				fbADSWRITE( WRITE:= FALSE );
				fbADSWRITE(
					NETID:= TcMcGlobal.NCNETID_TCMC,
					PORT:= AMSPORT_R0_NCSAF,
					IDXGRP:= 16#4200 + Axis.NcToPlc.AxisId,
					IDXOFFS:= 16#63,
					LEN:= SIZEOF(stWriteDriveOperationMode),
					SRCADDR:= ADR(stWriteDriveOperationMode),
					WRITE:= TRUE,
					TMOUT:= TcMcGlobal.tADSTimeOut);
				state := STATE_ORDER;
			END_IF
		END_IF

	STATE_ORDER :
		fbADSWRITE();
		IF NOT fbADSWRITE.BUSY THEN
			IF NOT fbADSWRITE.ERR THEN
				Done := TRUE;
			ELSE
				Error := TRUE;
				ErrorID := fbADSWRITE.ERRID;
			END_IF
			state := STATE_INITIALIZATION;
		END_IF

END_CASE

ADSbusy := fbADSWRITE.BUSY;
IF state = STATE_INITIALIZATION THEN
	(* reset Busy immediately  when sequence ends *)
	IF Busy THEN
		LastExecutionResult.Done := Done;
		LastExecutionResult.Error := Error;
		LastExecutionResult.ErrorID := ErrorID;
	END_IF
	Busy := FALSE;
END_IF

END_FUNCTION_BLOCK

// POUs/Administrative/Extensions/MC_CalcDynamicsByRampTime
FUNCTION_BLOCK MC_CalcDynamicsByRampTime
VAR_INPUT
	Velocity 	: LREAL;		// must be greaater than zero
	RampTime 	: LREAL;		// must be greaater than zero
	Stiffness 	: LREAL := 0.5;	// range 0..1.0 (will be silently reduced to 0.99 if 0.99 < Stiffness <= 1.0) 
END_VAR
VAR_OUTPUT
	Error 		: BOOL;
	ErrorID 	: UDINT;
	Acceleration: LREAL;	
	Deceleration: LREAL;	// identical to Acceleration !	
	Jerk 		: LREAL;
END_VAR
VAR
	t1: LREAL;	// time of jerk to ramp up to constant acceleration
	t2: LREAL;	// time of constant acceleration
	TriggerExecute: R_trig;
END_VAR

// Description:
//
// The function block calculates Acceleration and Jerk values to ramp up to a defined Velcoity in a defined RampTime.
// The calculation assumes that the Velocity can be reached (long distance moves). The calculated dynamics can be  
// used on short distances moves as well but the ramp up time will then be shorter. 
//
// Velocity : Velocity value to ramp up to during RampTime
// RampTime : time to ramp up to Velocity
// Stiffness: = time of constant acceleration / time to ramp up to constant acceleration (jerk time)
// 		Sample:  
// 			Stiffness = 0.0	: triangular acceleration profile
// 			Stiffness = 0.5	: trapezoid acceleration profile with time of constant acceleration = 1/3 RampTime
//			Stiffness = 1.0	: rectangular acceleration profile 

// check input parameters
IF stiffness<0 OR stiffness>1.0 OR RampTime<0.001 OR Velocity < 0.001 THEN
	// error
	Error := TRUE;
	ErrorID := MC_ERROR_PARAMETER_NOT_CORRECT;
	Acceleration := 0;
	Deceleration := 0;
	Jerk := 0;
	RETURN;
END_IF

// silent reduction of Stiffness between 0.99 and 1.0 
IF Stiffness > 0.99 THEN
	Stiffness:=0.99;
END_IF

// t1 = time of jerk to ramp up to constant acceleration
t1 := (1-Stiffness) / (2-Stiffness) * RampTime; 
(*
// check ?
IF t1<0.000250 THEN
	t1 := 0.000250;
END_IF
*)
// t2 = time of constant acceleration
t2 := RampTime - t1 - t1; // RampTime - 2*t1	

Acceleration := Velocity / (t1 + t2);
Deceleration := Acceleration;
Jerk := Acceleration / t1;

Error := FALSE; // result okay
ErrorID := 0;

END_FUNCTION_BLOCK

// POUs/Administrative/Extensions/MC_SelectControlLoop
{attribute 'conditionalshow_all_locals'}
FUNCTION_BLOCK MC_SelectControlLoop
VAR_IN_OUT
	Axis : AXIS_REF; (*Reference to an axis*)
END_VAR
VAR_INPUT
	Execute : BOOL;
	EncoderIndex : UINT;
	SelectType : E_SelectControlLoopType;
	SyncValue : LREAL;
	ExtSetPointGen : BOOL;
END_VAR
VAR_OUTPUT
	Done : BOOL;
	Busy : BOOL;
	Error : BOOL;
{attribute 'displaymode':='hex'}
	ErrorID : UDINT;
END_VAR
VAR
	LastExecutionResult: 	_ST_FunctionBlockResults;
	ADSbusy: BOOL;
	state: _E_TcMC_STATES := STATE_INITIALIZATION;
	stSelectControlLoop : ST_SelectControlLoop;
	fbADSWRITE: ADSWRITE;
END_VAR
VAR
	TriggerExecute: R_TRIG;
END_VAR

TriggerExecute(CLK:=Execute);

CASE state OF
	STATE_INITIALIZATION :
		Busy := FALSE;
		IF NOT Execute THEN
			Done := FALSE;
			Error := FALSE;
			ErrorID := 0;
		END_IF
		IF TriggerExecute.Q THEN
			Busy := TRUE;

			LastExecutionResult.Done := FALSE;
			LastExecutionResult.CommandAborted := FALSE;
			LastExecutionResult.Error := FALSE;
			LastExecutionResult.ErrorID := 0;
	
			stSelectControlLoop.EncoderIndex := EncoderIndex;
			stSelectControlLoop.SelectType := SelectType;
			stSelectControlLoop.SyncValue := SyncValue;
			stSelectControlLoop.ExtSetPointGen := SEL(ExtSetPointGen, 0 ,1);

			fbADSWRITE( WRITE:= FALSE );
			fbADSWRITE(
				NETID:= TcMcGlobal.NCNETID_TCMC,
				PORT:= TcMcGlobal.NCPORT_TCMC,
				IDXGRP:= 16#4200 + Axis.NcToPlc.AxisId,
				IDXOFFS:= 16#52,
				LEN:= SIZEOF(stSelectControlLoop),
				SRCADDR:= ADR(stSelectControlLoop),
				WRITE:= TRUE,
				TMOUT:= TcMcGlobal.tADSTimeOut);
			state := STATE_ORDER;
		END_IF

	STATE_ORDER :
		fbADSWRITE();
		IF NOT fbADSWRITE.BUSY THEN
			IF NOT fbADSWRITE.ERR THEN
				Done := TRUE;
			ELSE
				Error := TRUE;
				ErrorID := fbADSWRITE.ERRID;
			END_IF
			state := STATE_INITIALIZATION;
		END_IF

END_CASE

ADSbusy := fbADSWRITE.BUSY;
IF state = STATE_INITIALIZATION THEN
	(* reset Busy immediately  when sequence ends *)
	IF Busy THEN
		LastExecutionResult.Done := Done;
		LastExecutionResult.Error := Error;
		LastExecutionResult.ErrorID := ErrorID;
	END_IF
	Busy := FALSE;
END_IF

END_FUNCTION_BLOCK

// POUs/Administrative/Extensions/MC_WriteNcIoOutput
{attribute 'conditionalshow_all_locals'}
FUNCTION_BLOCK MC_WriteNcIoOutput
VAR_IN_OUT
	Axis				: AXIS_REF;
END_VAR
VAR_INPUT
	Execute				: BOOL;

	Device				: E_NcIoDevice := NcIoDeviceDrive;	
	NcIoOutput			: E_NcIoOutput := NcIoOutputnCtrl1;
	
	BitSelectMask		: UDINT := 16#0;
	BitValues			: UDINT;
END_VAR
VAR_OUTPUT
	Done				: BOOL;
	Busy				: BOOL;
	Error				: BOOL;
{attribute 'displaymode':='hex'}
	ErrorId				: UDINT;
END_VAR
VAR
	FlExecute			: R_TRIG;
	
	State				: UDINT;
	
	ReadDriveAddress	: MC_ReadDriveAddress;
	DriveAddress		: ST_DriveAddress;
	
	AdsWrite			: ADSWRITE;
	IdxGrp				: UDINT;

	NcIoOutputData		: _ST_NcIoOutputData;
END_VAR

FlExecute(CLK:=Execute);

CASE State OF
	0:
		IF NOT Execute THEN
			Done := FALSE;
			Busy := FALSE;
			Error := FALSE;
			ErrorId := 0;
		END_IF
		
		IF FlExecute.Q THEN
			Busy := TRUE;
			IF DriveAddress.NcAxisId = Axis.NcToPlc.AxisId THEN
				State := State + 2;
			ELSE
				State := State + 1;
			END_IF
		END_IF
		
	1: // Read drive address
		ReadDriveAddress(
			Axis			:= Axis, 
			Execute			:= TRUE, 
			DriveAddress	=> DriveAddress);

		IF NOT ReadDriveAddress.Busy AND ReadDriveAddress.Done THEN
			ReadDriveAddress(
				Axis			:= Axis, 
				Execute			:= FALSE); 

			State := State + 1	;		
		ELSIF NOT ReadDriveAddress.Busy AND ReadDriveAddress.Error THEN
			Busy := FALSE;
			Error := TRUE;
			ErrorId := ReadDriveAddress.ErrorID;
			
			ReadDriveAddress(
				Axis			:= Axis, 
				Execute			:= FALSE); 
				
			State := 0;	
		END_IF

	2: // Write nc io output
		CASE Device OF
			NcIoDeviceDrive:
				IdxGrp := 16#7300 + DriveAddress.NcDriveId;				
			NcIoDeviceEncoder:
				IdxGrp := 16#5300 + DriveAddress.NcEncoderId;				
			ELSE
				Busy := FALSE;
				Error := TRUE;
				ErrorId := 16#4B06;

				State := 0;
				RETURN;				
		END_CASE
	
		CASE NcIoOutput OF
			NcIoOutputnCtrl1:
				NcIoOutputData.ByteOffset := 16#08;
			NcIoOutputnCtrl2:
				NcIoOutputData.ByteOffset := 16#09;
			NcIoOutputnCtrl3:
				NcIoOutputData.ByteOffset := 16#0A;
			NcIoOutputnCtrl4:
				NcIoOutputData.ByteOffset := 16#0B;
			NcIoOutputnCtrl5:
				NcIoOutputData.ByteOffset := 16#1C;
			NcIoOutputnCtrl6:
				NcIoOutputData.ByteOffset := 16#1D;
			NcIoOutputnCtrl7:
				NcIoOutputData.ByteOffset := 16#1E;
			NcIoOutputnCtrl8:
				NcIoOutputData.ByteOffset := 16#1F;
			NcIoOutputnDataOut1:
				NcIoOutputData.ByteOffset := 16#00;
			NcIoOutputnDataOut2:
				NcIoOutputData.ByteOffset := 16#04;
			NcIoOutputnDataOut3:
				NcIoOutputData.ByteOffset := 16#0C;
			NcIoOutputnDataOut4:
				NcIoOutputData.ByteOffset := 16#10;
			NcIoOutputnDataOut5:
				NcIoOutputData.ByteOffset := 16#14;
			NcIoOutputnDataOut6:
				NcIoOutputData.ByteOffset := 16#18;
			ELSE			
				Busy := FALSE;
				Error := TRUE;
				ErrorId := 16#4B06;

				State := 0;
				RETURN;				
		END_CASE

		NcIoOutputData.BitSelectMask 	:= BitSelectMask;
		NcIoOutputData.BitValues		:= BitValues;

		AdsWrite(
			NETID			:= '', 
			PORT			:= 501, 
			IDXGRP			:= IdxGrp, 
			IDXOFFS			:= 16#01, 
			LEN				:= SIZEOF(NcIoOutputData), 
			SRCADDR			:= ADR(NcIoOutputData), 
			WRITE			:= TRUE, 
			TMOUT			:= T#5S); 

		IF AdsWrite.BUSY THEN
			State := State + 1;
		END_IF

	3: // wait for result
		AdsWrite();

		IF NOT AdsWrite.BUSY THEN
			IF NOT AdsWrite.ERR THEN
				Done := TRUE;				
			ELSE
				Error := TRUE;
				ErrorId := AdsWrite.ERRID;				
			END_IF
			Busy := FALSE;
			
			AdsWrite(WRITE := FALSE);
			
			State := 0;
		END_IF
END_CASE

END_FUNCTION_BLOCK

// POUs/Administrative/Status and Parameter/MC_ReadActualPosition
FUNCTION_BLOCK MC_ReadActualPosition
(*	This Function Block returns the actual position. *)
VAR_IN_OUT
	Axis			:	AXIS_REF; (*Reference to an axis*)
END_VAR
VAR_INPUT
	Enable		:	BOOL;		
END_VAR
VAR_OUTPUT
	Valid		:	BOOL;		
	Busy		:	BOOL;		
	Error		:	BOOL;	
{attribute 'displaymode':='hex'}
	ErrorID		:	UDINT;	
	Position		:	LREAL;		
END_VAR
VAR
END_VAR

Error := FALSE;
ErrorID := 0;
IF Enable THEN
	Busy := TRUE;
	Position := Axis.NcToPlc.ActPos;
	Valid := TRUE;
ELSE
	Busy := FALSE;
	Position := 0.0;
	Valid := FALSE;
END_IF;

END_FUNCTION_BLOCK

// POUs/Administrative/Status and Parameter/MC_ReadActualVelocity
FUNCTION_BLOCK MC_ReadActualVelocity
(*
	This Function Block returns the value of the actual velocity as long as Enable is 
	set. Valid is true when the data-output ActualVelocity is valid. If Enable is reset, the 
	data loses its validity, and all outputs are reset, no matter if new data is available.
*)
VAR_IN_OUT
	Axis			:	AXIS_REF; (*Reference to an axis*)
END_VAR
VAR_INPUT
	Enable 		: 	BOOL;	
END_VAR
VAR_OUTPUT
	Valid 		: 	BOOL;	
	Busy 		: 	BOOL;	
	Error 		: 	BOOL;	
{attribute 'displaymode':='hex'}
	ErrorID 		: 	UDINT;	
	ActualVelocity (* Velocity *): 	LREAL;	
END_VAR
VAR
END_VAR

Error := FALSE;
ErrorID := 0;
IF Enable THEN
	Busy := TRUE;
	Valid := TRUE;
	ActualVelocity := Axis.NcToPlc.ActVelo;
ELSE
	Busy := FALSE;
	Valid := FALSE;
	ActualVelocity := 0;
END_IF

END_FUNCTION_BLOCK

// POUs/Administrative/Status and Parameter/MC_ReadAxisError
FUNCTION_BLOCK MC_ReadAxisError
(*
	This Function Block presents general axis errors not relating to the Function Blocks. 
	(for instance axis errors, drive errors, communication errors)
 *)
VAR_IN_OUT
	Axis				:	AXIS_REF; (*Reference to an axis*)
END_VAR
VAR_INPUT
	Enable			:	BOOL;		
END_VAR
VAR_OUTPUT
	Valid			:	BOOL;		
	Busy			:	BOOL;		
	Error			:	BOOL;	
{attribute 'displaymode':='hex'}
	ErrorID			:	DWORD;	
	AxisErrorID		:	DWORD;	
END_VAR
VAR
END_VAR

IF Enable THEN
	Busy		 := TRUE;
	Valid 		:=  TRUE;
	ErrorID 		:= 0;
	AxisErrorID 	:= Axis.NcToPlc.ErrorCode;
	Error		:= ErrorID <> 0;
ELSE
	Busy 		:= FALSE;
	Valid 		:= FALSE;
	Error 		:= FALSE;	(* reset at falling edge of Execute *)
	ErrorID 		:= 0;
	AxisErrorID 	:= 0;
END_IF;

END_FUNCTION_BLOCK

// POUs/Administrative/Status and Parameter/MC_WriteBoolParameter
FUNCTION_BLOCK MC_WriteBoolParameter
(*	This Function Block modifies the value of a vendor specific boolean parameter. *)
VAR_IN_OUT
	Axis				:	AXIS_REF; (*Reference to an axis*)
END_VAR
VAR_INPUT
	Execute			:	BOOL;	
	ParameterNumber	:	MC_AxisParameter; // 2023-03 KSt changed from INT to MC_AxisParameter	
	Value			:	BOOL;	
(* 	ExecutionMode 	: 	MC_EXECUTION_MODE *)		(* not available *)
END_VAR
VAR_OUTPUT
	Done			:	BOOL;	
	Busy			: 	BOOL;
	Error			:	BOOL;	
{attribute 'displaymode':='hex'}
	ErrorID			:	UDINT;	
END_VAR
VAR
	ADSbusy		: 	BOOL;
	fbReadWriteParameter: 	_FB_ReadWriteParameter;
END_VAR
VAR
//{attribute 'conditionalshow'}
//	nParatype 		:	_E_ParameterType;	(* removed 2021-04-12 KSt - not required *)
{attribute 'conditionalshow'}
	dwValue 			: 	DWORD;
{attribute 'conditionalshow'}
	lrValue 			: 	LREAL;
{attribute 'conditionalshow'}
	fbTrigger 		: 	R_TRIG;
END_VAR

IF NOT Execute THEN
	Done := FALSE;
	Error := FALSE;			(* reset at falling edge of Execute *)
	ErrorID := 0;
END_IF
fbTrigger(CLK:= Execute);
IF fbTrigger.Q AND NOT Busy THEN
	Busy := TRUE;
	Done := FALSE;
	Error := FALSE;
	ErrorID := MC_ERROR_NO_ERROR;
END_IF;
(* *)
IF Busy THEN
//	nParatype := PARAMETERTYPE_BOOL;
	fbReadWriteParameter.ParameterPointer := 0;
	fbReadWriteParameter.ParameterSize := 0;
	fbReadWriteParameter(Enable:= TRUE, ParameterNumber:= ParameterNumber, Mode:= READWRITEPARAMETERMODE_WRITE,
						(*ParameterType:=nParatype,*) Axis:= Axis, ValueLreal:= lrValue, ValueDword := dwValue, ValueBool := Value);
	IF fbReadWriteParameter.Done THEN
		Done := TRUE;
		Busy := FALSE;
		fbReadWriteParameter(Enable:= FALSE, ParameterNumber:= ParameterNumber, Mode:= READWRITEPARAMETERMODE_WRITE,
						(*ParameterType:= nParatype,*) Axis:= Axis, ValueLreal:= lrValue, ValueDword := dwValue, ValueBool := Value);
	END_IF;
	IF fbReadWriteParameter.Error THEN
		Busy := FALSE;
		Done := FALSE;
		Error := TRUE;
		ErrorID := fbReadWriteParameter.ErrorID;
		fbReadWriteParameter(Enable:= FALSE, ParameterNumber:= ParameterNumber, Mode:= READWRITEPARAMETERMODE_WRITE,
						(*ParameterType:= nParatype,*) Axis:= Axis, ValueLreal:= lrValue, ValueDword := dwValue, ValueBool := Value);
	END_IF;
END_IF;

ADSbusy := fbReadWriteParameter.ADSbusy;

END_FUNCTION_BLOCK

// POUs/Administrative/Status and Parameter/MC_WriteLargeParameter
FUNCTION_BLOCK MC_WriteLargeParameter
(*	This Function Block modifies the value of a vendor specific parameter. *)
VAR_IN_OUT
	Axis				:	AXIS_REF; (*Reference to an axis*)
END_VAR
VAR_INPUT
	Execute			:	BOOL;	
	ParameterNumber	:	MC_AxisParameter; // 2023-03 KSt changed from INT to MC_AxisParameter		
//	Value			:	LREAL;	
	ParameterPointer: 	PVOID;	// for structured parameters - KSt 2021-03-04
	ParameterSize	:	USINT; 	// for structured parameters  - KSt 2021-03-04
(* 	ExecutionMode 	: 	MC_EXECUTION_MODE *)	(* not available *)
END_VAR
VAR_OUTPUT
	Done			:	BOOL;		
	Busy			: 	BOOL;		
	Error			:	BOOL;		
{attribute 'displaymode':='hex'}
	ErrorID			:	UDINT;		
END_VAR
VAR
	ADSbusy			: 	BOOL;
	fbReadWriteParameter: _FB_ReadWriteParameter;
END_VAR
VAR
{attribute 'conditionalshow'}
	lrValue 		: 	LREAL;
{attribute 'conditionalshow'}
	dwValue 		: 	DWORD;
{attribute 'conditionalshow'}
	bValue 			: 	BOOL;
{attribute 'conditionalshow'}
	fbTrigger 		: 	R_TRIG;
END_VAR

IF NOT Execute THEN
	Done := FALSE;
	Error := FALSE;			(* reset at falling edge of Execute *)
	ErrorID := 0;
END_IF
fbTrigger(CLK:= Execute);
IF fbTrigger.Q AND NOT Busy THEN
	Busy := TRUE;
	Done := FALSE;
	Error := FALSE;
	ErrorID := MC_ERROR_NO_ERROR;
END_IF;
(* *)
IF Busy THEN
	fbReadWriteParameter.ParameterPointer := 0;
	fbReadWriteParameter.ParameterSize := 0;
	fbReadWriteParameter(Enable:= TRUE, ParameterNumber:= ParameterNumber, Mode:= READWRITEPARAMETERMODE_WRITE,
						Axis:= Axis, ValueLreal:= lrValue, ValueDword := dwValue, ValueBool := bValue,
						ParameterPointer := ParameterPointer, ParameterSize:=ParameterSize); 
	IF fbReadWriteParameter.Done THEN
		Done := TRUE;
		Busy := FALSE;
		fbReadWriteParameter(Enable:= FALSE, ParameterNumber:= ParameterNumber, Mode:= READWRITEPARAMETERMODE_WRITE,
							Axis:= Axis, ValueLreal:= lrValue, ValueDword := dwValue, ValueBool := bValue,
							ParameterPointer := ParameterPointer, ParameterSize:=ParameterSize); 
	END_IF;
	IF fbReadWriteParameter.Error THEN
		Busy := FALSE;
		Done := FALSE;
		Error := TRUE;
		ErrorID := fbReadWriteParameter.ErrorID;
		fbReadWriteParameter(Enable:= FALSE, ParameterNumber:= ParameterNumber, Mode:= READWRITEPARAMETERMODE_WRITE,
							Axis:= Axis, ValueLreal:= lrValue, ValueDword := dwValue, ValueBool := bValue,
							ParameterPointer := ParameterPointer, ParameterSize:=ParameterSize); 
	END_IF;
END_IF;

ADSbusy := fbReadWriteParameter.ADSbusy;

END_FUNCTION_BLOCK

// POUs/Administrative/Status and Parameter/MC_WriteLargeParameterPersistent
FUNCTION_BLOCK MC_WriteLargeParameterPersistent
VAR_IN_OUT
	Axis: AXIS_REF; (*Reference to an axis*)
END_VAR
VAR_INPUT
	Execute			: BOOL;
	ParameterNumber	: MC_AxisParameter; // 2023-03 KSt changed from INT to MC_AxisParameter
//	Value: LREAL;
	ParameterPointer: 	PVOID;	// for structured parameters - KSt 2021-03-04
	ParameterSize	:	USINT; 	// for structured parameters  - KSt 2021-03-04
END_VAR
VAR_OUTPUT
	Done: BOOL;
	Busy: BOOL;
	Error: BOOL;
{attribute 'displaymode':='hex'}
	ErrorID: UDINT;
END_VAR
VAR
	fbWriteParameterPersistent: _FB_WriteParameterPersistent;
END_VAR

fbWriteParameterPersistent(
	Axis:= Axis, 
	Execute:= Execute, 
	ParameterNumber:= ParameterNumber, 
//	Value:= Value, 
	ParameterPointer := ParameterPointer, 
	ParameterSize:=ParameterSize,
	Done=> Done, 
	Busy=> Busy, 
	Error=> Error, 
	ErrorID=> ErrorID);

END_FUNCTION_BLOCK

// POUs/Motion/Phasing/MC_HaltPhasing
FUNCTION_BLOCK MC_HaltPhasing
VAR_IN_OUT
	Master 			: 	AXIS_REF; (*Reference to an axis*)
	Slave 			: 	AXIS_REF; (*Reference to an axis*)
END_VAR
VAR_INPUT
	Execute			:	BOOL;		(* Start the motion at rising edge *)
	Deceleration	:	LREAL;		(* Value of the maximum deceleration *)
	Jerk			:	LREAL;		(* Value of the maximum jerk *)
	BufferMode		:	MC_BufferMode;	
	Options			: 	ST_PhasingOptions;		(* optional parameters *)
END_VAR
VAR_OUTPUT
	Done			:	BOOL;	
	Busy			: 	BOOL;	
	Active			: 	BOOL;	
	CommandAborted	:	BOOL;	
	Error			:	BOOL;	
{attribute 'displaymode':='hex'}
	ErrorID			:	UDINT;	
END_VAR

VAR
	PhasingGeneric : _FB_PhasingGeneric;
END_VAR

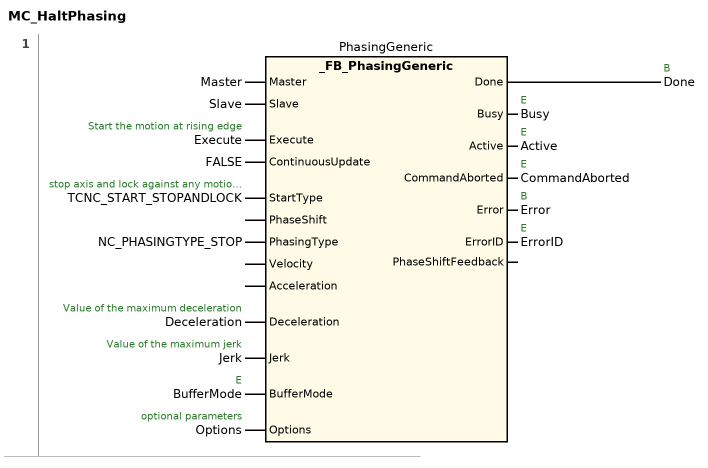
// NETWORK 1
//   Execute: Start the motion at rising edge
//   TCNC_START_STOPANDLOCK: stop axis and lock against any motion commands
//   Deceleration: Value of the maximum deceleration
//   Jerk: Value of the maximum jerk
//   BufferMode: E
//   Options: optional parameters
//   Busy: E
//   Active: E
//   CommandAborted: E
//   Error: B
//   ErrorID: E
//   Done: B
PhasingGeneric(
    Master := Master,
    Slave := Slave,
    Execute := Execute,
    ContinuousUpdate := FALSE,
    StartType := TCNC_START_STOPANDLOCK,
    PhasingType := NC_PHASINGTYPE_STOP,
    Deceleration := Deceleration,
    Jerk := Jerk,
    BufferMode := BufferMode,
    Options := Options,
    Busy => Busy,
    Active => Active,
    CommandAborted => CommandAborted,
    Error => Error,
    ErrorID => ErrorID); // _FB_PhasingGeneric
Done := PhasingGeneric.Done;

END_FUNCTION_BLOCK

// POUs/Motion/Phasing/MC_PhasingAbsolute
(*	This Function Block creates an absolute phase shift in the master position of a slave axis. 
	The master position is shifted in relation to the real physical position. This is analogous 
	to opening a coupling on the master shaft for a moment, and is used to delay or advance 
	an axis to its master. The phase shift is seen from the slave. The master does not know 
	that there is a phase shift experienced by the slave (MasterPos as seen from the 
	SlaveAxis = PhysicalMasterPos + PhaseShiftValueSlaveAxis, the phase shift value has 
	the character of a position offset) The phase shift remains until another Phasing 
	command changes it again. *)
FUNCTION_BLOCK MC_PhasingAbsolute
VAR_IN_OUT
	Master 			: 	AXIS_REF; (*Reference to an axis*)
	Slave 			: 	AXIS_REF; (*Reference to an axis*)
END_VAR
VAR_INPUT
	Execute			:	BOOL;		(* Start the motion at rising edge *)
	ContinuousUpdate:	BOOL; (* changes for PhaseShift, Velocity, Acceleration, Deceleration and Jekr can be updated while command is executing *)
	PhaseShift		:	LREAL;		(* Target position for the motion *)
	Velocity		:	LREAL;		(* Value of the maximum velocity *)
	Acceleration	:	LREAL;		(* Value of the maximum acceleration *)
	Deceleration	:	LREAL;		(* Value of the maximum deceleration *)
	Jerk			:	LREAL;		(* Value of the maximum jerk *)
	BufferMode		:	MC_BufferMode;		
	Options			: 	ST_PhasingOptions;		(* optional parameters *)
END_VAR
VAR_OUTPUT
	Done			:	BOOL;	
	Busy			: 	BOOL;	
	Active			: 	BOOL;	
	CommandAborted	:	BOOL;	
	Error			:	BOOL;	
{attribute 'displaymode':='hex'}
	ErrorID			:	UDINT;	
	AbsolutePhaseShift : 	LREAL;	
END_VAR

VAR
	PhasingGeneric : _FB_PhasingGeneric;
END_VAR

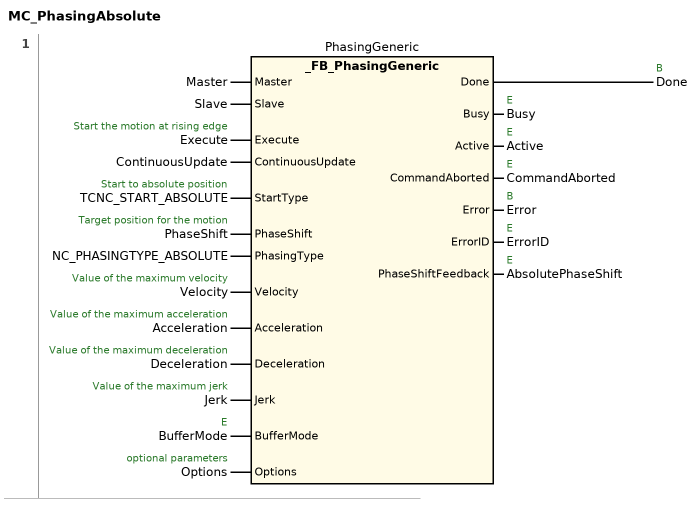
// NETWORK 1
//   Execute: Start the motion at rising edge
//   TCNC_START_ABSOLUTE: Start to absolute position
//   PhaseShift: Target position for the motion
//   Velocity: Value of the maximum velocity
//   Acceleration: Value of the maximum acceleration
//   Deceleration: Value of the maximum deceleration
//   Jerk: Value of the maximum jerk
//   BufferMode: E
//   Options: optional parameters
//   Busy: E
//   Active: E
//   CommandAborted: E
//   Error: B
//   ErrorID: E
//   AbsolutePhaseShift: E
//   Done: B
PhasingGeneric(
    Master := Master,
    Slave := Slave,
    Execute := Execute,
    ContinuousUpdate := ContinuousUpdate,
    StartType := TCNC_START_ABSOLUTE,
    PhaseShift := PhaseShift,
    PhasingType := NC_PHASINGTYPE_ABSOLUTE,
    Velocity := Velocity,
    Acceleration := Acceleration,
    Deceleration := Deceleration,
    Jerk := Jerk,
    BufferMode := BufferMode,
    Options := Options,
    Busy => Busy,
    Active => Active,
    CommandAborted => CommandAborted,
    Error => Error,
    ErrorID => ErrorID,
    PhaseShiftFeedback => AbsolutePhaseShift); // _FB_PhasingGeneric
Done := PhasingGeneric.Done;

END_FUNCTION_BLOCK

// POUs/Motion/Phasing/MC_PhasingRelative
(*	This Function Block creates a phase shift in the master position of a slave axis relative 
	to the existing phase shift.
	The master position is shifted in relation to the real physical position. This is analogous 
	to opening a coupling on the master shaft for a moment, and is used to delay or advance 
	an axis to its master. The phase shift is seen from the slave. The master does not know 
	that there is a phase shift experienced by the slave. (MasterPos as seen from 
	SlaveAxis = PhysicalMasterPos + PhaseShiftValueSlaveAxis, the phase shift value has 
	the character of a position offset) The phase shift remains until another Phasing 
	command changes it again. Relative phase shifts are added to each other for the 
	applicable phase shift. *)
FUNCTION_BLOCK MC_PhasingRelative
VAR_IN_OUT
	Master 			: 	AXIS_REF; (*Reference to an axis*)
	Slave 			: 	AXIS_REF; (*Reference to an axis*)
END_VAR
VAR_INPUT
	Execute			:	BOOL;	(* Start the motion at rising edge *)
	ContinuousUpdate:	BOOL;	(* changes for PhaseShift, Velocity, Acceleration, Deceleration and Jekr can be updated while command is executing *)
	PhaseShift		:	LREAL;	(* Target position for the motion *)
	Velocity		:	LREAL;	(* Value of the maximum velocity *)
	Acceleration	:	LREAL;	(* Value of the maximum acceleration *)
	Deceleration	:	LREAL;	(* Value of the maximum deceleration *)
	Jerk			:	LREAL;	(* Value of the maximum jerk *)
	BufferMode		:	MC_BufferMode;		
	Options			: 	ST_PhasingOptions;	(* optional parameters *)
END_VAR
VAR_OUTPUT
	Done			:	BOOL;	
	Busy			: 	BOOL;	
	Active			: 	BOOL;	
	CommandAborted	:	BOOL;	
	Error			:	BOOL;	
{attribute 'displaymode':='hex'}
	ErrorID			:	UDINT;	
	CoveredPhaseShift : 	LREAL;	
END_VAR

VAR
	PhasingGeneric : _FB_PhasingGeneric;
END_VAR

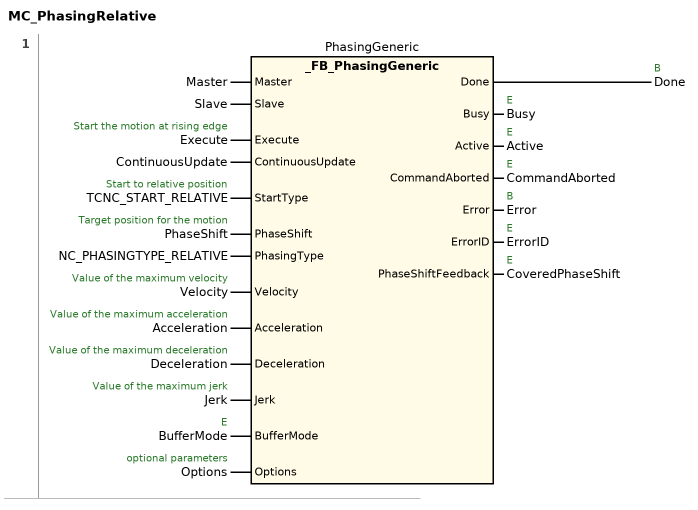
// NETWORK 1
//   Execute: Start the motion at rising edge
//   TCNC_START_RELATIVE: Start to relative position
//   PhaseShift: Target position for the motion
//   Velocity: Value of the maximum velocity
//   Acceleration: Value of the maximum acceleration
//   Deceleration: Value of the maximum deceleration
//   Jerk: Value of the maximum jerk
//   BufferMode: E
//   Options: optional parameters
//   Busy: E
//   Active: E
//   CommandAborted: E
//   Error: B
//   ErrorID: E
//   CoveredPhaseShift: E
//   Done: B
PhasingGeneric(
    Master := Master,
    Slave := Slave,
    Execute := Execute,
    ContinuousUpdate := ContinuousUpdate,
    StartType := TCNC_START_RELATIVE,
    PhaseShift := PhaseShift,
    PhasingType := NC_PHASINGTYPE_RELATIVE,
    Velocity := Velocity,
    Acceleration := Acceleration,
    Deceleration := Deceleration,
    Jerk := Jerk,
    BufferMode := BufferMode,
    Options := Options,
    Busy => Busy,
    Active => Active,
    CommandAborted => CommandAborted,
    Error => Error,
    ErrorID => ErrorID,
    PhaseShiftFeedback => CoveredPhaseShift); // _FB_PhasingGeneric
Done := PhasingGeneric.Done;

END_FUNCTION_BLOCK

// POUs/Motion/Point To Point Motion/MC_MoveContinuousAbsolute
FUNCTION_BLOCK MC_MoveContinuousAbsolute
(*	This function block commands a controlled motion to a specified absolute position
	ending with the specified velocity.

	Notes:
	- If the target is reached and no new motion command is put into the buffer, the 
	  axis continues to run with the specified EndVelocity.
	- This Function Block places the axis into the 'Continuous Motion' state, even 
	  during the initial motion by a relative distance, and remains in the 'Continuous 
	  Motion' state once the EndVelocity has been reached.
	- This FB can be replaced by the combination of MC_MoveAbsolute and 
	  MC_MoveVelocity

	MoveContinous ist ähnlich MoveVelocity. Es wird aber zunächst mit einem PTP-Profil
	eine Zwischenposition angefahren (mit Velocity). Ab dieser Position geht die Bewegung
	in eine Endlosfahrt mit EndVelocity über.
*)
VAR_IN_OUT
	Axis				:	AXIS_REF; (*Reference to an axis*)
END_VAR
VAR_INPUT
	Execute			:	BOOL;	
(*	ContinuousUpdate :	BOOL; *)		(* not available *)
	Position			:	LREAL;	
	Velocity			:	LREAL;	
	EndVelocity		:	LREAL;	
	Acceleration		:	LREAL;	
	Deceleration		:	LREAL;	
	Jerk				:	LREAL;	
(*	Direction 		:	MC_Direction;	*)		(* not available *)
	BufferMode		:	MC_BufferMode;	
	Options			: 	ST_MoveOptions;
END_VAR
VAR_OUTPUT
	InEndVelocity	:	BOOL;	
	Busy			: 	BOOL;	
	Active			: 	BOOL;	
	CommandAborted :	BOOL;	
	Error			:	BOOL;	
{attribute 'displaymode':='hex'}
	ErrorID			:	UDINT;	
END_VAR
VAR
	LastExecutionResult: 	_ST_FunctionBlockResults;
	ADSbusy		: 	BOOL;
	MoveGeneric		: 	_FB_MoveUniversalGeneric;
	CmdNo: UINT;
END_VAR

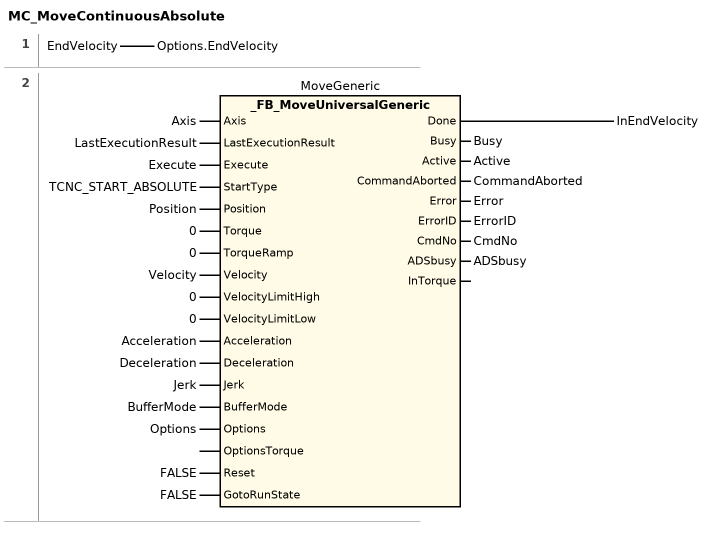
// NETWORK 1
Options.EndVelocity := EndVelocity;

// NETWORK 2
MoveGeneric(
    Axis := Axis,
    LastExecutionResult := LastExecutionResult,
    Execute := Execute,
    StartType := TCNC_START_ABSOLUTE,
    Position := Position,
    Torque := 0,
    TorqueRamp := 0,
    Velocity := Velocity,
    VelocityLimitHigh := 0,
    VelocityLimitLow := 0,
    Acceleration := Acceleration,
    Deceleration := Deceleration,
    Jerk := Jerk,
    BufferMode := BufferMode,
    Options := Options,
    Reset := FALSE,
    GotoRunState := FALSE,
    Busy => Busy,
    Active => Active,
    CommandAborted => CommandAborted,
    Error => Error,
    ErrorID => ErrorID,
    CmdNo => CmdNo,
    ADSbusy => ADSbusy); // _FB_MoveUniversalGeneric
InEndVelocity := MoveGeneric.Done;

END_FUNCTION_BLOCK

// POUs/Motion/Point To Point Motion/MC_MoveContinuousRelative
FUNCTION_BLOCK MC_MoveContinuousRelative
(*	This function block commands a controlled motion of a specified relative distance
	ending with the specified velocity.

	Notes:
	- If the target is reached and no new motion command is put into the buffer, the 
	  axis continues to run with the specified EndVelocity.
	- This Function Block places the axis into the 'Continuous Motion' state, even 
	  during the initial motion by a relative distance, and remains in the 'Continuous 
	  Motion' state once the EndVelocity has been reached.
 	- This FB can be replaced by the combination of MC_MoveRelative and 
	  MC_MoveVelocity 

	MoveContinous ist ähnlich MoveVelocity. Es wird aber zunächst mit einem PTP-Profil
	eine Zwischenposition angefahren (mit Velocity). Ab dieser Position geht die Bewegung
	in eine Endlosfahrt mit EndVelocity über.
*)
VAR_IN_OUT
	Axis				:	AXIS_REF; (*Reference to an axis*)
END_VAR
VAR_INPUT
	Execute			:	BOOL;	
(*	ContinuousUpdate :	BOOL; *)		(* not available *)
	Distance			:	LREAL;	
	Velocity			:	LREAL;	
	EndVelocity		:	LREAL;	
	Acceleration		:	LREAL;	
	Deceleration		:	LREAL;	
	Jerk				:	LREAL;	
	BufferMode		:	MC_BufferMode;	
	Options			: 	ST_MoveOptions;
END_VAR
VAR_OUTPUT
	InEndVelocity		:	BOOL;	
	Busy			: 	BOOL;	
	Active			: 	BOOL;	
	CommandAborted :	BOOL;	
	Error			:	BOOL;	
{attribute 'displaymode':='hex'}
	ErrorID			:	UDINT;	
END_VAR
VAR
	LastExecutionResult: 	_ST_FunctionBlockResults;
	ADSbusy		: 	BOOL;
	MoveGeneric		: 	_FB_MoveUniversalGeneric;
	CmdNo: UINT;
END_VAR

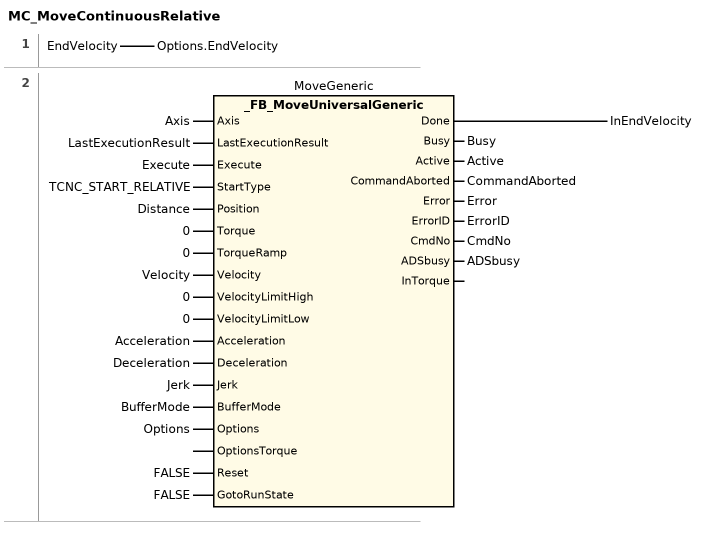
// NETWORK 1
Options.EndVelocity := EndVelocity;

// NETWORK 2
MoveGeneric(
    Axis := Axis,
    LastExecutionResult := LastExecutionResult,
    Execute := Execute,
    StartType := TCNC_START_RELATIVE,
    Position := Distance,
    Torque := 0,
    TorqueRamp := 0,
    Velocity := Velocity,
    VelocityLimitHigh := 0,
    VelocityLimitLow := 0,
    Acceleration := Acceleration,
    Deceleration := Deceleration,
    Jerk := Jerk,
    BufferMode := BufferMode,
    Options := Options,
    Reset := FALSE,
    GotoRunState := FALSE,
    Busy => Busy,
    Active => Active,
    CommandAborted => CommandAborted,
    Error => Error,
    ErrorID => ErrorID,
    CmdNo => CmdNo,
    ADSbusy => ADSbusy); // _FB_MoveUniversalGeneric
InEndVelocity := MoveGeneric.Done;

END_FUNCTION_BLOCK

// POUs/Motion/Torque Control/MC_TorqueControl
{attribute 'conditionalshow_all_locals'}
FUNCTION_BLOCK MC_TorqueControl
VAR_IN_OUT
	Axis						: AXIS_REF;
END_VAR
VAR_INPUT
	Execute						: BOOL;
	ContinuousUpdate			: BOOL;
	Relative					: BOOL;
	Torque						: LREAL; // [%]
	TorqueRamp					: LREAL; // [%/s]
	VelocityLimitHigh			: LREAL;
	VelocityLimitLow			: LREAL;
	BufferMode					: MC_BufferMode := MC_BufferMode.MC_Aborting; 
	Options						: ST_TorqueControlOptions;
END_VAR
VAR_OUTPUT
	InTorque					: BOOL;
	Busy						: BOOL;
	Active						: BOOL;
	CommandAborted				: BOOL;
	Error						: BOOL;
{attribute 'displaymode':='hex'}
	ErrorId						: UDINT;
END_VAR
VAR
	LastExecutionResult			: 	_ST_FunctionBlockResults;
	ADSbusy						: 	BOOL;
	MoveGeneric					: 	_FB_MoveUniversalGeneric;
	CmdNo						: UINT;
END_VAR

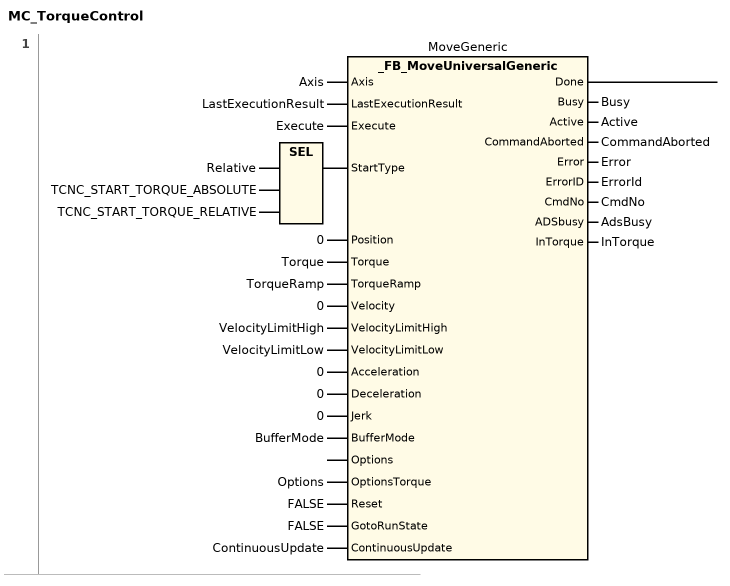
// NETWORK 1
MoveGeneric(
    Axis := Axis,
    LastExecutionResult := LastExecutionResult,
    Execute := Execute,
    StartType := SEL(Relative, TCNC_START_TORQUE_ABSOLUTE, TCNC_START_TORQUE_RELATIVE),
    Position := 0,
    Torque := Torque,
    TorqueRamp := TorqueRamp,
    Velocity := 0,
    VelocityLimitHigh := VelocityLimitHigh,
    VelocityLimitLow := VelocityLimitLow,
    Acceleration := 0,
    Deceleration := 0,
    Jerk := 0,
    BufferMode := BufferMode,
    OptionsTorque := Options,
    Reset := FALSE,
    GotoRunState := FALSE,
    ContinuousUpdate := ContinuousUpdate,
    Busy => Busy,
    Active => Active,
    CommandAborted => CommandAborted,
    Error => Error,
    ErrorID => ErrorId,
    CmdNo => CmdNo,
    ADSbusy => AdsBusy,
    InTorque => InTorque); // _FB_MoveUniversalGeneric

END_FUNCTION_BLOCK
